TYPE Storage :
STRUCT
	Component: STRING;
	Quatity: INT;
END_STRUCT
END_TYPE

(* stored: Version 1.1.0.1, ProductVersion 3.1.4022.16
   DUT Storage: Id {b8019088-7461-4c6d-b793-eaf619a7cf86} *)
